// TIA Portal V15.1 export
// export: Created 2020-06-12T07:35:45.4130859Z, ExportSetting None, DisplayName Totally Integrated Automation Portal, DisplayVersion V15.1, DisplayName TIA Portal Openness, DisplayVersion V15.1, DisplayName STEP 7 Professional, DisplayVersion V15.1, DisplayName STEP 7 Safety, DisplayVersion V15.1, DisplayName WinCC Advanced, DisplayVersion V15.1
FUNCTION "Alloy_call" : Void   // FC159, FBD
TITLE = Alloy addition call
{ S7_Optimized_Access := 'TRUE' }
// stored: SetENOAutomatically False
BEGIN

REGION Network 1
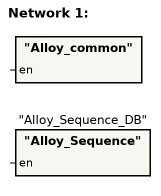
   "Alloy_common"();
   "Alloy_Sequence_DB"();   // "Alloy_Sequence"
END_REGION
END_FUNCTION
